INTERFACE I_TcpDevice

PROPERTY Active : REFERENCE TO BOOL
GET
END_GET
END_PROPERTY

PROPERTY AmsNetId : T_IPv4Addr
GET
END_GET
SET
END_SET
END_PROPERTY

PROPERTY Error : REFERENCE TO BOOL
GET
END_GET
END_PROPERTY

PROPERTY ErrorID : REFERENCE TO UDINT
GET
END_GET
END_PROPERTY

PROPERTY Host : T_IPv4Addr
GET
END_GET
SET
END_SET
END_PROPERTY

PROPERTY LastRecivedMessage : ST_TcpBufferData
GET
END_GET
END_PROPERTY

METHOD MR_Abort : BOOL
VAR_INPUT
END_VAR
END_METHOD

METHOD MR_FirstCycle : BOOL
VAR_INPUT
	sName 		: STRING;		(*  *)
	sHost		: T_IPv4Addr;	(*  *)
	sAmsNetID	: T_AmsNetID;	(*  *)
	iPort		: UINT;			(*  *)
	tTimeout	: TIME;			(*  *)
END_VAR
END_METHOD

METHOD MR_Init : BOOL
VAR_INPUT
END_VAR
END_METHOD

PROPERTY NextRecivedMessage : ST_TcpBufferData
GET
END_GET
END_PROPERTY

PROPERTY Port : UINT
GET
END_GET
SET
END_SET
END_PROPERTY

PROPERTY State : REFERENCE TO E_TcpIpDeviceState
GET
END_GET
END_PROPERTY

PROPERTY Timeout : TIME
GET
END_GET
SET
END_SET
END_PROPERTY

END_INTERFACE

(* stored: Version 1.1.0.1, ProductVersion 3.1.4024.12
   Itf I_TcpDevice: Id {24641fed-fe0c-4c17-ac00-6a81e0cb7f9a}
   Property Active: Id {e6e78939-3bec-453c-94fd-ceb2da17de4b}
   Get Get: Id {eed37a80-1f58-4113-9cfc-79cd624c49d5}
   Property AmsNetId: Id {f3c16fe1-985d-4794-92fc-0553d5d26b52}
   Get Get: Id {ad05585d-a341-44ea-833c-9638feff184d}
   Set Set: Id {2dab40f5-d94b-44b8-8920-4c58e4d3cf65}
   Property Error: Id {18b96bbc-5ddc-4554-9767-c3856f1495c8}
   Get Get: Id {1eb3bc57-f6b3-4078-9247-def055dbdf6f}
   Property ErrorID: Id {75c8d22c-5b3d-4aca-b038-2efc9b31e3b5}
   Get Get: Id {e67f7001-ed6f-4197-8d5d-2e93cd3f31a2}
   Property Host: Id {e8bc6caa-ba3c-49fe-b1ae-321f66c6df87}
   Get Get: Id {e040dc30-5927-4fdb-9bc5-daff8d153b56}
   Set Set: Id {4406a13c-44da-4e2b-928a-3e793c107a24}
   Property LastRecivedMessage: Id {3798787f-9098-460b-b8af-f91d765d2507}
   Get Get: Id {b2610185-8255-458b-97a9-4b59bd498eb3}
   Method MR_Abort: Id {769cd83c-40db-4fb2-aebc-dd8ea19ebb89}
   Method MR_FirstCycle: Id {cf8eacf6-dc9a-4f90-9f0e-4234ff6db895}
   Method MR_Init: Id {4583fa0a-1fb6-41d4-adb2-4edf06982c1d}
   Property NextRecivedMessage: Id {1093f905-dd34-4788-8088-36459b46f8ff}
   Get Get: Id {bdf418df-7520-465d-bb35-f8dbe577629f}
   Property Port: Id {f541c0e6-0474-4220-b6e1-fa5c3a040faa}
   Get Get: Id {2ea7bed2-0e99-459b-978e-f586ac4ca061}
   Set Set: Id {a1982a94-5dd5-4134-8c57-f27831474b14}
   Property State: Id {d2bc7920-f576-46c7-a2a1-841f510b29cd}
   Get Get: Id {bf49696b-3bc0-47ff-ab8e-49a575a61d3b}
   Property Timeout: Id {1816e9d4-9944-4fc6-a56f-05dde3353985}
   Get Get: Id {4157fa2d-cc8c-4fef-92e8-3476043ac959}
   Set Set: Id {93014aca-0db0-4bcb-a462-30cc1c18e385} *)
